// Mitsubishi GX Works2 project: EX2   PLC: FX3G

// global labels: Global1
VAR_GLOBAL
  CreamInput AT D1111 : REAL;
  CreamInput1 AT D2 : REAL;
  inputtttt AT D1 : REAL;
  CreamQuantity AT D1113 : REAL;
END_VAR
VAR_GLOBAL CONSTANT
  MinCream : REAL := 300;
END_VAR
VAR_GLOBAL
  Lamp7 AT Y007 : BOOL;
  StartDay AT X007 : BOOL;
  ChocolateInput AT D1115 : REAL;
  BiscuitInput AT D1119 : REAL;
  ChocolateQuantity AT D1117 : REAL;
  BiscuitQuantity AT D1121 : REAL;
END_VAR
VAR_GLOBAL CONSTANT
  MinBiscuit : REAL := 6;
  MinChocolate : REAL := 240;
END_VAR
VAR_GLOBAL
  MovingCream AT X011 : BOOL;
  Lamp2 AT Y002 : BOOL;
  Label0 AT M0 : BOOL;
  Switch1 AT X001 : BOOL;
  Out1 AT TS1 : BOOL;
  Lamp0 AT Y000 : BOOL;
  AAAA AT TC2 : BOOL;
  Out2 AT TS2 : BOOL;
  Lamp1 AT Y001 : BOOL;
  Lamp3 AT Y003 : BOOL;
  Timer4 AT TC3 : BOOL;
END_VAR
VAR_GLOBAL CONSTANT
  FourSeconds : INT := 40;
END_VAR
VAR_GLOBAL
  Out3 AT TS3 : BOOL;
  Label1 AT M1 : BOOL;
  Timer1 AT TC1 : BOOL;
END_VAR
VAR_GLOBAL CONSTANT
  Sec : INT := 1;
END_VAR
VAR_GLOBAL
  Timer2 AT TC2 : BOOL;
  StartZiluf AT X010 : BOOL;
  Switch6 AT X006 : BOOL;
  Analog1 AT D8280 : INT;
  AnalogVal AT D8201 : INT;
END_VAR
VAR_GLOBAL CONSTANT
  Five : INT := 2100;
  SmallCoating : REAL := 120;
  DoubleCoating : REAL := 240;
END_VAR
VAR_GLOBAL
  Label3 AT M3 : BOOL;
  Label15 AT M15 : BOOL;
END_VAR
VAR_GLOBAL CONSTANT
  Fghdfgh : INT := 16800;
END_VAR
VAR_GLOBAL
  Label14 AT M14 : BOOL;
  EndDay AT M10 : BOOL;
  Timer5 AT TC5 : BOOL;
END_VAR
VAR_GLOBAL CONSTANT
  FiveSec : INT := 50;
END_VAR
VAR_GLOBAL
  Out5 AT TS5 : BOOL;
  Label16 AT M16 : BOOL;
  Switch0 AT X000 : BOOL;
  Counter1 AT CC1 : BOOL;
END_VAR
VAR_GLOBAL CONSTANT
  CountingToFive : WORD := 5;
END_VAR
VAR_GLOBAL
  OutC1 AT CS1 : BOOL;
  Counter2 AT CC2 : BOOL;
END_VAR
VAR_GLOBAL CONSTANT
  CountingToSix : WORD := 6;
END_VAR
VAR_GLOBAL
  OutC2 AT CS2 : BOOL;
  Creambo AT D1139 : REAL;
  CreamboQuantity AT D1141 : REAL;
END_VAR
VAR_GLOBAL CONSTANT
  SixCreambo : REAL := 238;
END_VAR
VAR_GLOBAL
  AnalogOutPut AT D8282 : INT;
  Label17 AT M17 : BOOL;
  Counter3 AT CC3 : BOOL;
  OutC3 AT CS3 : BOOL;
  Timer6 AT TC6 : BOOL;
END_VAR
VAR_GLOBAL CONSTANT
  ThreeSec : INT := 30;
END_VAR
VAR_GLOBAL
  Label7 AT M7 : BOOL;
  Timer7 AT TC7 : BOOL;
  Out7 AT TS7 : BOOL;
  Timer8 AT TC8 : BOOL;
  Out8 AT TS8 : BOOL;
  Label8 AT M8 : BOOL;
  Label9 AT M9 : BOOL;
  Out66 AT TS6 : BOOL;
  AlmostEnd AT M20 : BOOL;
  Label19 AT M19 : BOOL;
  CreamboInt AT D1143 : INT;
  Label20 AT M50 : BOOL;
  Label21 AT M21 : BOOL;
  EndOfZiluf AT M100 : BOOL;
  EndOfCoating AT M101 : BOOL;
  HoldLamp3 AT M102 : BOOL;
END_VAR
VAR_GLOBAL CONSTANT
  ThreeHundredCream : REAL := 300;
END_VAR
VAR_GLOBAL
  Ziluf AT D1200 : REAL;
END_VAR
VAR_GLOBAL CONSTANT
  Zero : REAL;
END_VAR
VAR_GLOBAL
  TurnOnMachineA AT X010 : BOOL;
  MachineA AT M40 : BOOL;
  Sen_Cam AT X001 : BOOL;
  Sen_Touch AT M42 : BOOL;
  ErrorSwitch AT X005 : BOOL;
  Sen_30 AT X003 : BOOL;
  Sen_15 AT X002 : BOOL;
  Lamp4 AT Y004 : BOOL;
  LuckOfCream AT M45 : BOOL;
  LuckOfChoc AT M46 : BOOL;
  LuckOfBisquit AT M47 : BOOL;
  HoldLamp4 AT M91 : BOOL;
  ReadyToZiluf AT M81 : BOOL;
  Empty AT M82 : BOOL;
  Diping AT D1205 : REAL;
  ReadyToDip AT M82 : BOOL;
END_VAR

// task Task_01 (event TRUE, interval 0, priority 31): POU_01

PROGRAM POU_01
VAR
  Out6 : BOOL;
END_VAR
(* structured ladder/FBD written out as ST: instructions are called as NAME(EN, inputs, outputs); _pN, _eN, _tN stand for wires *)
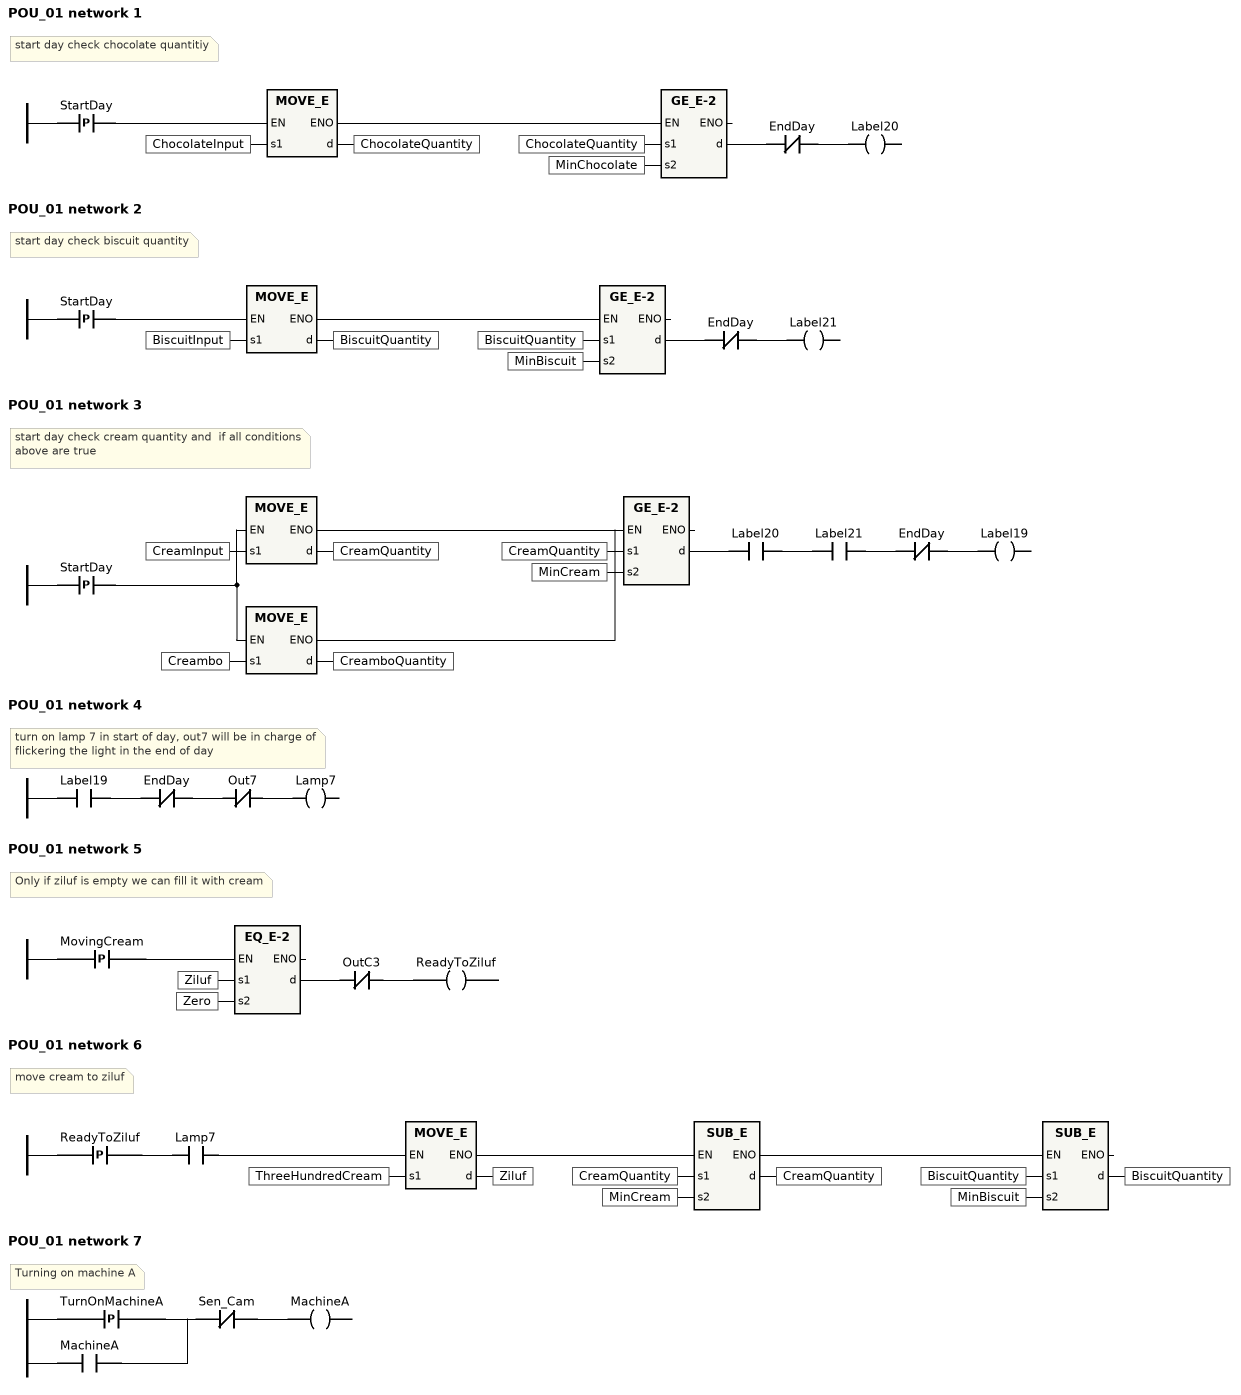
(* network 1 *)
(* start day check chocolate quantitiy *)
_e1 := MOVE_E(LDP(TRUE, StartDay), ChocolateInput, ChocolateQuantity);
GE_E(_e1, ChocolateQuantity, MinChocolate, _t2);
Label20 := _t2 AND NOT EndDay;
(* network 2 *)
(* start day check biscuit quantity *)
_e1 := MOVE_E(LDP(TRUE, StartDay), BiscuitInput, BiscuitQuantity);
GE_E(_e1, BiscuitQuantity, MinBiscuit, _t2);
Label21 := _t2 AND NOT EndDay;
(* network 3 *)
(* start day check cream quantity and  if all conditions above are true *)
_p1 := LDP(TRUE, StartDay);
_e2 := MOVE_E(_p1, CreamInput, CreamQuantity);
_e3 := MOVE_E(_p1, Creambo, CreamboQuantity);
GE_E(_e2 OR _e3, CreamQuantity, MinCream, _t4);
Label19 := _t4 AND Label20 AND Label21 AND NOT EndDay;
(* network 4 *)
(* turn on lamp 7 in start of day, out7 will be in charge of flickering the light in the end of day *)
Lamp7 := Label19 AND NOT EndDay AND NOT Out7;
(* network 5 *)
(* Only if ziluf is empty we can fill it with cream *)
EQ_E(LDP(TRUE, MovingCream), Ziluf, Zero, _t1);
ReadyToZiluf := _t1 AND NOT OutC3;
(* network 6 *)
(* move cream to ziluf *)
_e1 := MOVE_E(LDP(TRUE, ReadyToZiluf) AND Lamp7, ThreeHundredCream, Ziluf);
_e2 := SUB_E(_e1, CreamQuantity, MinCream, CreamQuantity);
SUB_E(_e2, BiscuitQuantity, MinBiscuit, BiscuitQuantity);
(* network 7 *)
(* Turning on machine A *)
MachineA := (LDP(TRUE, TurnOnMachineA) OR MachineA) AND NOT Sen_Cam;
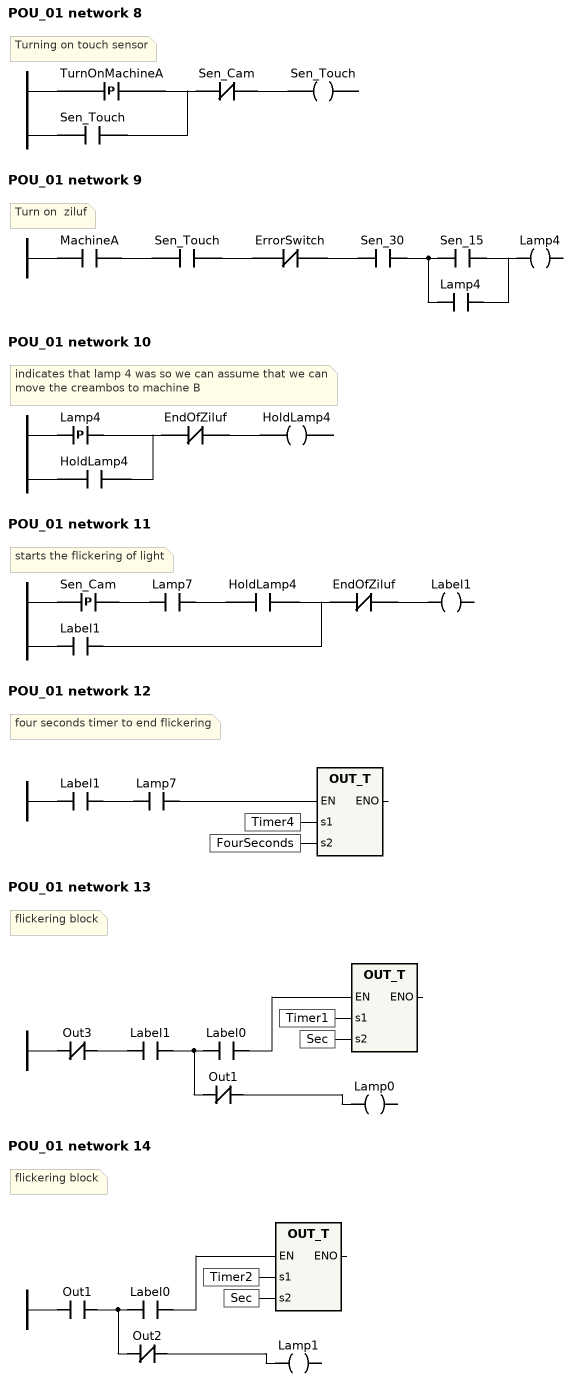
(* network 8 *)
(* Turning on touch sensor *)
Sen_Touch := (LDP(TRUE, TurnOnMachineA) OR Sen_Touch) AND NOT Sen_Cam;
(* network 9 *)
(* Turn on  ziluf *)
_p1 := MachineA AND Sen_Touch AND NOT ErrorSwitch AND Sen_30;
Lamp4 := (_p1 AND Sen_15) OR (_p1 AND Lamp4);
(* network 10 *)
(* indicates that lamp 4 was so we can assume that we can move the creambos to machine B *)
HoldLamp4 := (LDP(TRUE, Lamp4) OR HoldLamp4) AND NOT EndOfZiluf;
(* network 11 *)
(* starts the flickering of light *)
Label1 := ((LDP(TRUE, Sen_Cam) AND Lamp7 AND HoldLamp4) OR Label1) AND NOT EndOfZiluf;
(* network 12 *)
(* four seconds timer to end flickering *)
OUT_T(Label1 AND Lamp7, Timer4, FourSeconds);
(* network 13 *)
(* flickering block *)
_p1 := NOT Out3 AND Label1;
OUT_T(_p1 AND Label0, Timer1, Sec);
Lamp0 := _p1 AND NOT Out1;
(* network 14 *)
(* flickering block *)
OUT_T(Out1 AND Label0, Timer2, Sec);
Lamp1 := Out1 AND NOT Out2;
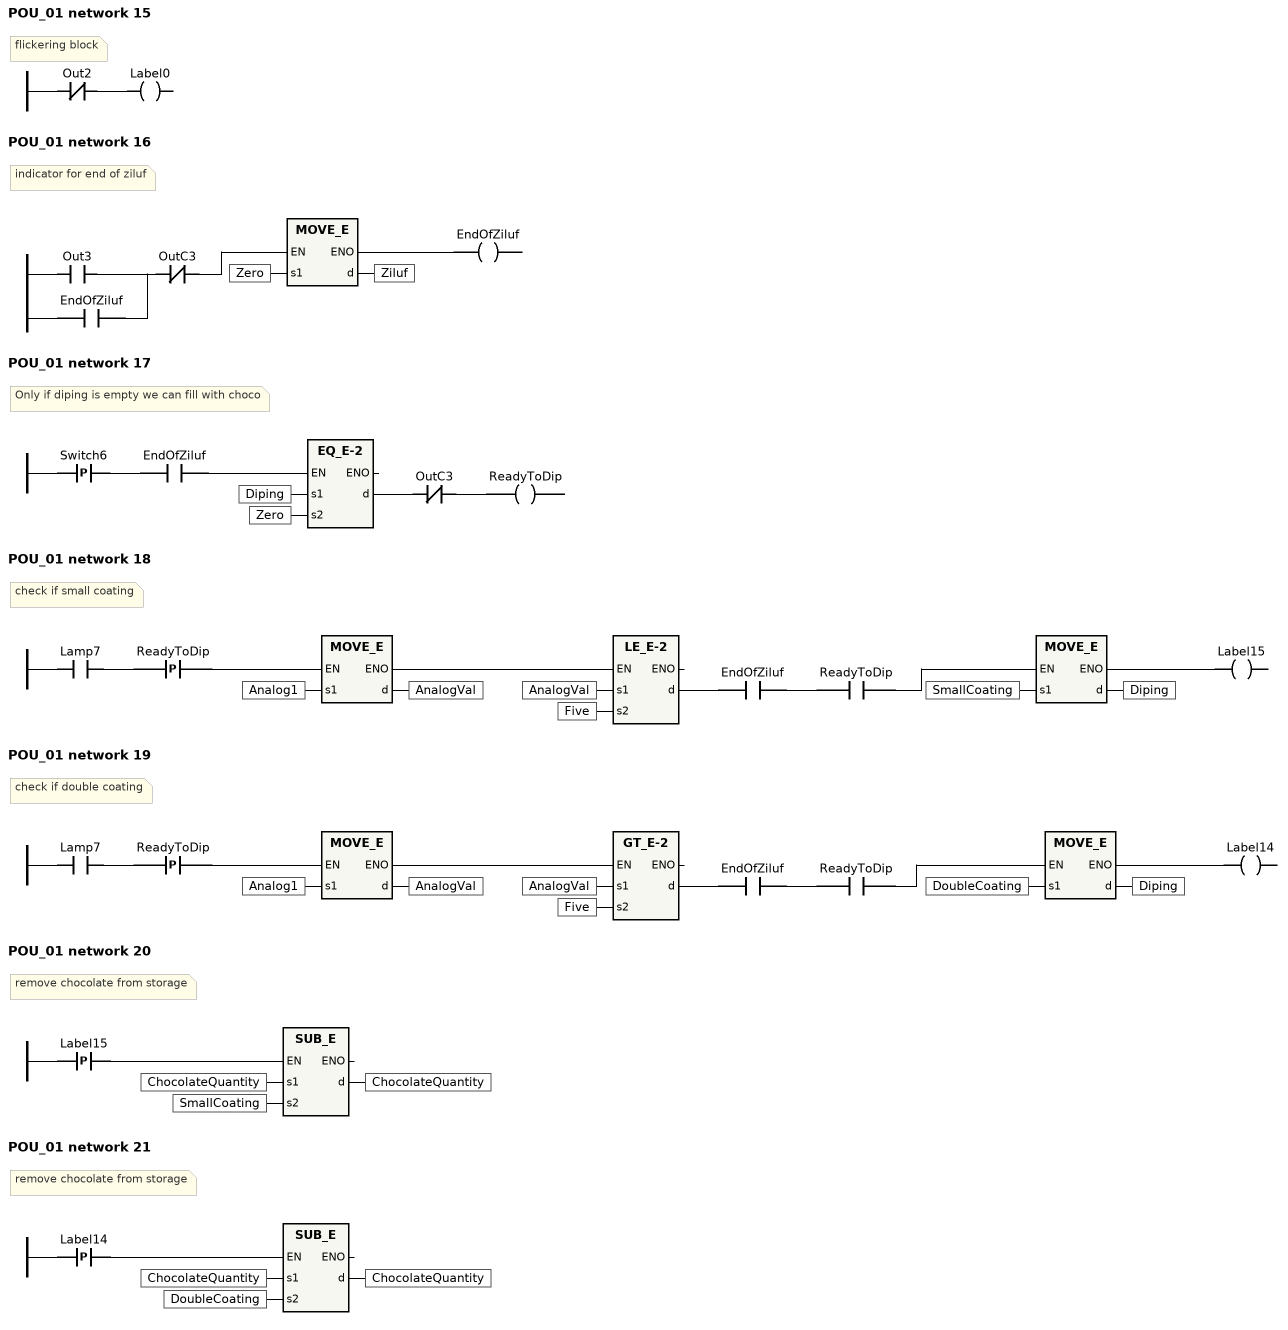
(* network 15 *)
(* flickering block *)
Label0 := NOT Out2;
(* network 16 *)
(* indicator for end of ziluf *)
_e1 := MOVE_E((Out3 OR EndOfZiluf) AND NOT OutC3, Zero, Ziluf);
EndOfZiluf := _e1;
(* network 17 *)
(* Only if diping is empty we can fill with choco *)
EQ_E(LDP(TRUE, Switch6) AND EndOfZiluf, Diping, Zero, _t1);
ReadyToDip := _t1 AND NOT OutC3;
(* network 18 *)
(* check if small coating *)
_e1 := MOVE_E(Lamp7 AND LDP(TRUE, ReadyToDip), Analog1, AnalogVal);
LE_E(_e1, AnalogVal, Five, _t2);
_e3 := MOVE_E(_t2 AND EndOfZiluf AND ReadyToDip, SmallCoating, Diping);
Label15 := _e3;
(* network 19 *)
(* check if double coating *)
_e1 := MOVE_E(Lamp7 AND LDP(TRUE, ReadyToDip), Analog1, AnalogVal);
GT_E(_e1, AnalogVal, Five, _t2);
_e3 := MOVE_E(_t2 AND EndOfZiluf AND ReadyToDip, DoubleCoating, Diping);
Label14 := _e3;
(* network 20 *)
(* remove chocolate from storage *)
SUB_E(LDP(TRUE, Label15), ChocolateQuantity, SmallCoating, ChocolateQuantity);
(* network 21 *)
(* remove chocolate from storage *)
SUB_E(LDP(TRUE, Label14), ChocolateQuantity, DoubleCoating, ChocolateQuantity);
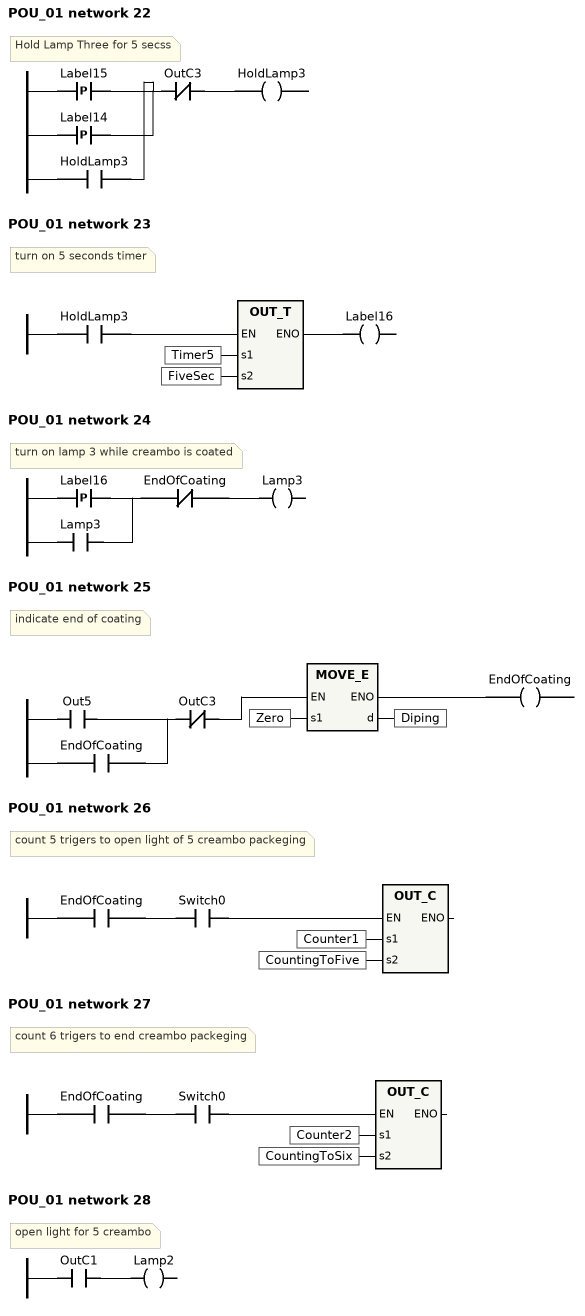
(* network 22 *)
(* Hold Lamp Three for 5 secss *)
HoldLamp3 := (LDP(TRUE, Label15) OR LDP(TRUE, Label14) OR HoldLamp3) AND NOT OutC3;
(* network 23 *)
(* turn on 5 seconds timer *)
_e1 := OUT_T(HoldLamp3, Timer5, FiveSec);
Label16 := _e1;
(* network 24 *)
(* turn on lamp 3 while creambo is coated *)
Lamp3 := (LDP(TRUE, Label16) OR Lamp3) AND NOT EndOfCoating;
(* network 25 *)
(* indicate end of coating *)
_e1 := MOVE_E((Out5 OR EndOfCoating) AND NOT OutC3, Zero, Diping);
EndOfCoating := _e1;
(* network 26 *)
(* count 5 trigers to open light of 5 creambo packeging *)
OUT_C(EndOfCoating AND Switch0, Counter1, CountingToFive);
(* network 27 *)
(* count 6 trigers to end creambo packeging *)
OUT_C(EndOfCoating AND Switch0, Counter2, CountingToSix);
(* network 28 *)
(* open light for 5 creambo *)
Lamp2 := OutC1;
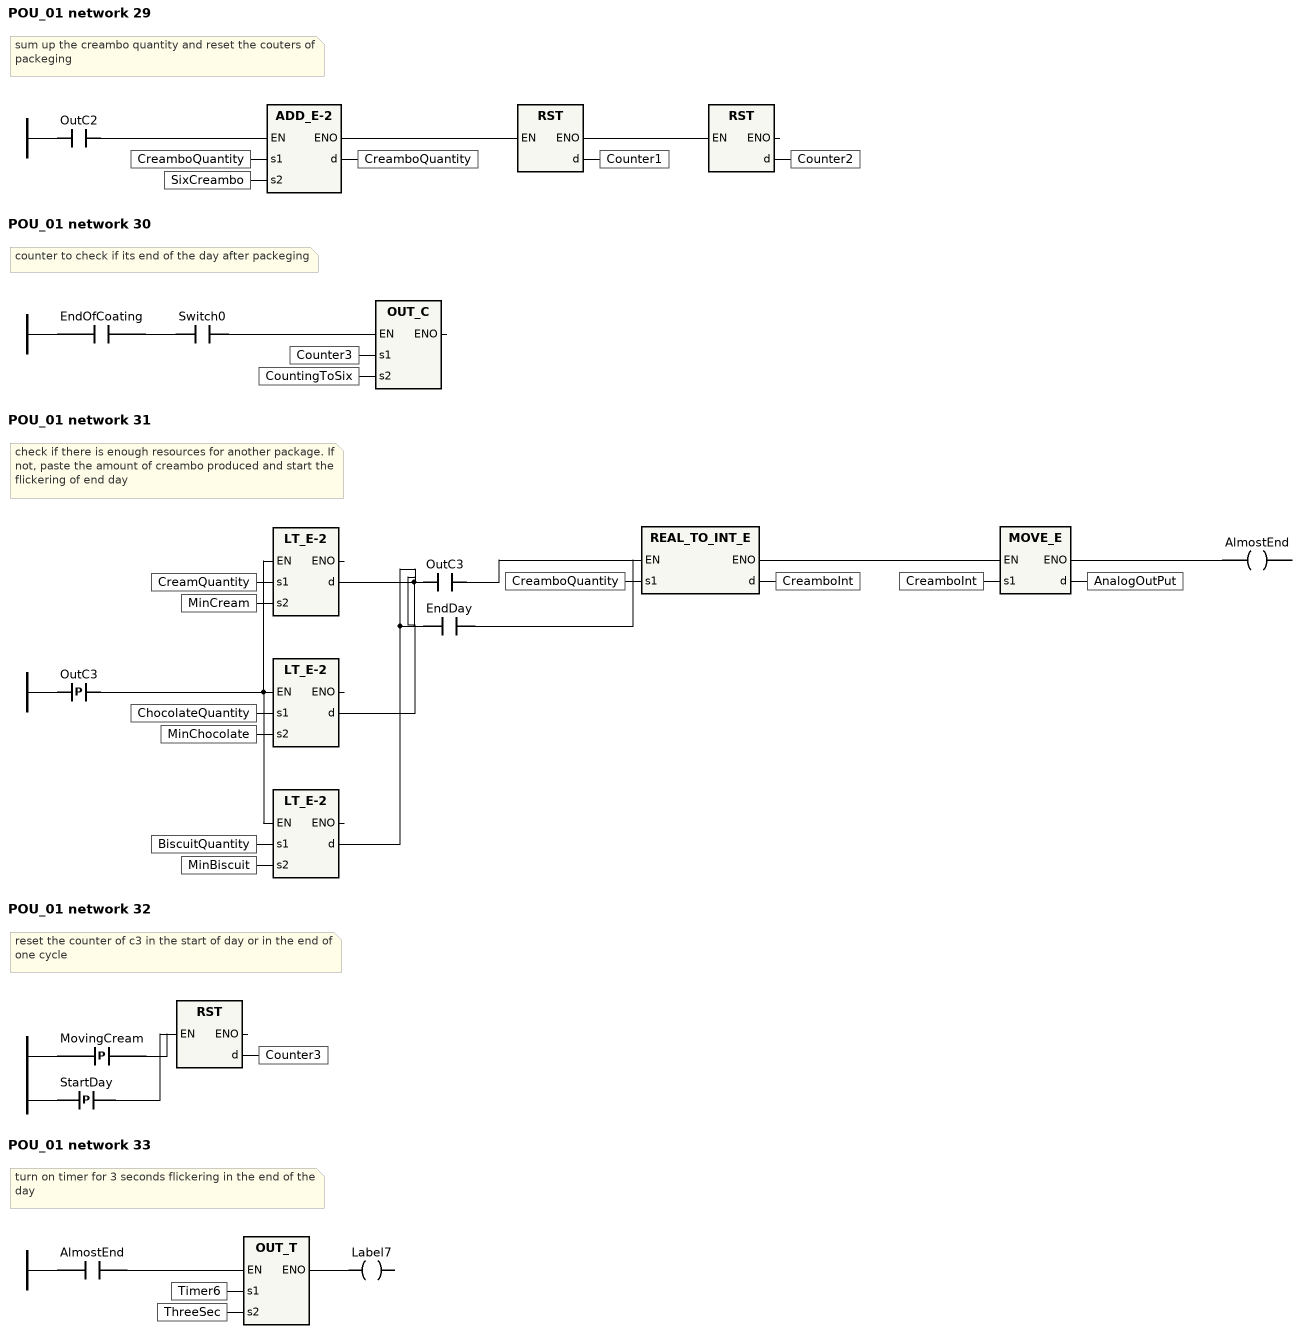
(* network 29 *)
(* sum up the creambo quantity and reset the couters of packeging *)
_e1 := ADD_E(OutC2, CreamboQuantity, SixCreambo, CreamboQuantity);
_e2 := RST(_e1, Counter1);
RST(_e2, Counter2);
(* network 30 *)
(* counter to check if its end of the day after packeging *)
OUT_C(EndOfCoating AND Switch0, Counter3, CountingToSix);
(* network 31 *)
(* check if there is enough resources for another package. If not, paste the amount of creambo produced and start the flickering of end day *)
_p1 := LDP(TRUE, OutC3);
LT_E(_p1, CreamQuantity, MinCream, _t2);
LT_E(_p1, ChocolateQuantity, MinChocolate, _t3);
LT_E(_p1, BiscuitQuantity, MinBiscuit, _t4);
_p5 := _t2 OR _t3 OR _t4;
_e6 := REAL_TO_INT_E((_p5 AND OutC3) OR (_p5 AND EndDay), CreamboQuantity, CreamboInt);
_e7 := MOVE_E(_e6, CreamboInt, AnalogOutPut);
AlmostEnd := _e7;
(* network 32 *)
(* reset the counter of c3 in the start of day or in the end of one cycle *)
RST(LDP(TRUE, MovingCream) OR LDP(TRUE, StartDay), Counter3);
(* network 33 *)
(* turn on timer for 3 seconds flickering in the end of the day *)
_e1 := OUT_T(AlmostEnd, Timer6, ThreeSec);
Label7 := _e1;
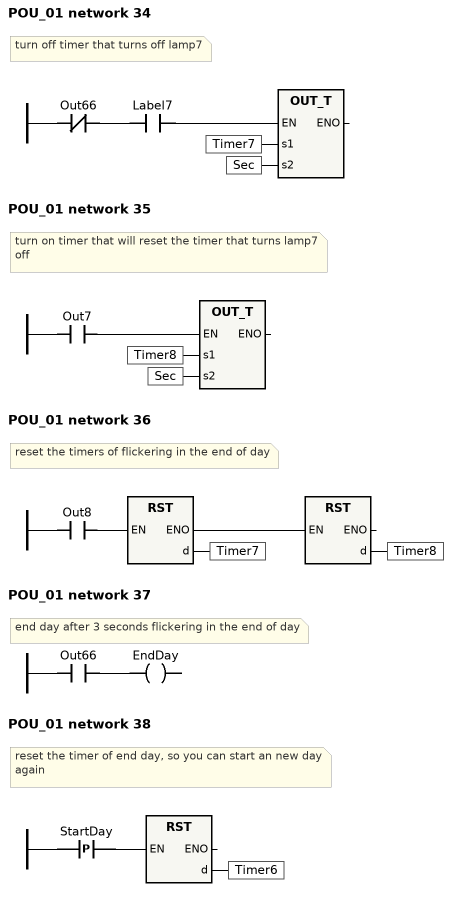
(* network 34 *)
(* turn off timer that turns off lamp7 *)
OUT_T(NOT Out66 AND Label7, Timer7, Sec);
(* network 35 *)
(* turn on timer that will reset the timer that turns lamp7 off *)
OUT_T(Out7, Timer8, Sec);
(* network 36 *)
(* reset the timers of flickering in the end of day *)
_e1 := RST(Out8, Timer7);
RST(_e1, Timer8);
(* network 37 *)
(* end day after 3 seconds flickering in the end of day *)
EndDay := Out66;
(* network 38 *)
(* reset the timer of end day, so you can start an new day again *)
RST(LDP(TRUE, StartDay), Timer6);
END_PROGRAM
